Fanuc KAREL source: kt00598.KL

-- PROVISIONAL review KL for V770-1; original PC SHA256 7bdf6d7fc68d8d4657c3eaeb88b988a51e239f51b5e80c2aaf0b784e9349207c
-- Incomplete behavior may be omitted. Consult companion uncertainty JSON. Do not deploy.
PROGRAM KT00598
%NOLOCKGROUP
VAR
  I1 : INTEGER
  I2 : INTEGER
  OUT : INTEGER
BEGIN
  -- UNRESOLVED_PC offsets 5-16; opcodes 2E,23
  -- UNRESOLVED_PC offsets 21-32; opcodes 2E,23
  -- UNRESOLVED_PC offsets 37-48; opcodes 2E,23
  -- UNRESOLVED_PC offsets 53-64; opcodes 2E,23
  -- UNRESOLVED_PC offsets 69-82; opcodes 21,48,23
  -- UNRESOLVED_PC offsets 87-91; opcodes 7F
END KT00598
